{attribute addProperty BoxType "EM7004-0000-0017"}
{attribute addProperty Id "Enable_PLSBIT10.1251"}
{attribute addProperty CRC "2222261065"}
{attribute addProperty SizeInBites "16"}
{attribute addProperty SizeInBytes "2"}
TYPE Control_84750349 :
STRUCT
	{attribute addProperty Name "Enable_PLS"}
	Enable_PLS : BIT;
	{attribute 'hide'}
	reserve_1_BIT_0 : BIT;
	{attribute 'hide'}
	reserve_1_BIT_1 : BIT;
	{attribute 'hide'}
	reserve_1_BIT_2 : BIT;
	{attribute 'hide'}
	reserve_1_BIT_3 : BIT;
	{attribute 'hide'}
	reserve_1_BIT_4 : BIT;
	{attribute 'hide'}
	reserve_1_BIT_5 : BIT;
	{attribute 'hide'}
	reserve_1_BIT_6 : BIT;
	{attribute 'hide'}
	reserve_1_BIT_7 : BIT;
	{attribute 'hide'}
	reserve_1_BIT_8 : BIT;
	{attribute 'hide'}
	reserve_1_BIT_9 : BIT;
	{attribute 'hide'}
	reserve_1_BIT_10 : BIT;
	{attribute 'hide'}
	reserve_1_BIT_11 : BIT;
	{attribute 'hide'}
	reserve_1_BIT_12 : BIT;
	{attribute 'hide'}
	reserve_1_BIT_13 : BIT;
	{attribute 'hide'}
	reserve_1_BIT_14 : BIT;
END_STRUCT
END_TYPE

(* stored: Version 1.2.0.0, ProductVersion 3.1.4024.9
   DUT Control_84750349: Id {1a5f5825-b7f2-4d72-ade0-8340fc53ecc4} *)
